// Monitors the chiller loop from the flow sensor
FUNCTION_BLOCK FB_ChillerLoop
VAR_INPUT
	bLoopTempSW : BOOL; // NC Temperature switch. Indicates when temperature is too high
END_VAR
VAR_OUTPUT
	{attribute 'pytmc' := '
		pv: ERROR
		io: i
		field: OSV MAJOR
		field: ZSV NO_ALARM
		field: ZNAM OK
		field: ONAM ERROR
	'}
	bError : BOOL := FALSE; // Whether an error was detected. Goes back to normal on its own
	{attribute 'pytmc' := '
		pv: OVERRIDE
		io: io
		field: ZNAM "OFF"
		field: ONAM "ON"
	'}
	bOperatorOverride : BOOL := FALSE; // If TRUE, allows the EPS to keep running despite the chiller loop error
END_VAR

(* Set error flag if loop temperature monitor detects an error *)
bError := NOT bLoopTempSW;

(* Reset the operator override if the system returns to normal tempreature range *)
IF bLoopTempSW THEN
	bOperatorOverride := FALSE;
END_IF

END_FUNCTION_BLOCK

(* stored: Version 1.1.0.1, ProductVersion 3.1.4024.6
   POU FB_ChillerLoop: Id {cb022f1c-3c99-48a7-a062-7a11524de8ff}, SpecialFunc None *)
